// TIA Portal V15.1 export
// export: Created 2024-06-21T08:40:58.8620848Z, ExportSetting WithDefaults, DisplayName Totally Integrated Automation Portal, DisplayVersion V15.1 Update 5, DisplayName TIA Portal Openness, DisplayVersion V15.1 Update 5, DisplayName SINAMICS Startdrive Advanced, DisplayVersion V15.1, DisplayName G130, G150, S120, S150, SINAMICS MV, S210, DisplayVersion V15.1, DisplayName G110M, G120, G120C, G120D, G120P, DisplayVersion V15.1, DisplayName STEP 7 Professional, DisplayVersion V15.1 Update 5, DisplayName STEP 7 Safety, DisplayVersion V15.1, DisplayName WinCC Professional, DisplayVersion V15.1 Update 5, DisplayName SIMATIC Visualization Architect, DisplayVersion V15.1
FUNCTION_BLOCK "LPNIODiagNameS7-1500"   // FB2213, SCL
{ S7_Optimized_Access := 'TRUE' }
VERSION : 0.1
// stored: AutoNumber false, IsIECCheckEnabled false, IsRetainMemResEnabled false, MemoryReserve 100, SetENOAutomatically False, UDAEnableTagReadback false
   VAR_INPUT
      I_StartFillList { ExternalAccessible := 'False'; ExternalVisible := 'False'; ExternalWritable := 'False'} : Bool;
      I_LastDeviceNumber { ExternalAccessible := 'False'; ExternalVisible := 'False'; ExternalWritable := 'False'} : Int;   // Last Device of ProfiNet System
      I_HWIOSYSTEM { ExternalAccessible := 'False'; ExternalVisible := 'False'; ExternalWritable := 'False'} : HW_IOSYSTEM;   // HW ID ProfiNet System
   END_VAR
   VAR_OUTPUT
      O_Done { ExternalAccessible := 'False'; ExternalVisible := 'False'; ExternalWritable := 'False'} : Bool;
      O_Name { ExternalAccessible := 'False'; ExternalVisible := 'False'; ExternalWritable := 'False'} : Array[0..255] of String[25];
   END_VAR
   VAR_IN_OUT
      IO_DeviceExist : Array[0..255] of Bool;   // IO devices exist
      IO_GetStationName : Array[0..255] of String;   // Profinet Name
   END_VAR
   VAR
      Index { ExternalAccessible := 'False'; ExternalVisible := 'False'; ExternalWritable := 'False'} : Int;
      LastDeviceNumber { ExternalAccessible := 'False'; ExternalVisible := 'False'; ExternalWritable := 'False'} : Int;   // Last Device of ProfiNet System
      Done { ExternalAccessible := 'False'; ExternalVisible := 'False'; ExternalWritable := 'False'} : Bool;
      DoneDelay { ExternalAccessible := 'False'; ExternalVisible := 'False'; ExternalWritable := 'False'} : Bool;
      ReturnGetNameBusy { ExternalAccessible := 'False'; ExternalVisible := 'False'; ExternalWritable := 'False'} : Bool;   // Temp
      ReturnGetNameDone { ExternalAccessible := 'False'; ExternalVisible := 'False'; ExternalWritable := 'False'} : Bool;   // Temp
      ReturnGetNameError { ExternalAccessible := 'False'; ExternalVisible := 'False'; ExternalWritable := 'False'} : Bool;   // Temp
      ReturnGetNameLen { ExternalAccessible := 'False'; ExternalVisible := 'False'; ExternalWritable := 'False'} : DInt;   // Temp
      ReturnGetNameStatus { ExternalAccessible := 'False'; ExternalVisible := 'False'; ExternalWritable := 'False'} : Word;   // Temp
      GetNameInstance { ExternalAccessible := 'False'; ExternalVisible := 'False'; ExternalWritable := 'False'; S7_SetPoint := 'True'} : Get_Name;   // Get Name of Devices
      TimerDone { ExternalAccessible := 'False'; ExternalVisible := 'False'; ExternalWritable := 'False'; S7_SetPoint := 'True'} : TON_TIME;
      EdgeStartFillList { ExternalAccessible := 'False'; ExternalVisible := 'False'; ExternalWritable := 'False'; S7_SetPoint := 'True'} : R_TRIG;
   END_VAR
BEGIN
   #EdgeStartFillList(CLK := #I_StartFillList);

   IF #EdgeStartFillList.Q THEN
       #Done := False;
       #Index := 0;
   END_IF;

   #LastDeviceNumber := #I_LastDeviceNumber;
   IF #I_LastDeviceNumber < 1 THEN
       #LastDeviceNumber := 1;
   END_IF;
   IF #I_LastDeviceNumber > 254 THEN
       #LastDeviceNumber := 254;
   END_IF;


   #TimerDone(IN := #Done,
              PT := T#500ms,
              Q => #DoneDelay);

   IF (#I_StartFillList & NOT #Done) THEN
       #Index := #Index + 1;
       IF #IO_DeviceExist[#Index] THEN
           WHILE (#IO_DeviceExist[#Index] & NOT #ReturnGetNameDone) DO
               #GetNameInstance(LADDR := #I_HWIOSYSTEM,
                    STATION_NR := INT_TO_UINT(#Index),
                    DONE => #ReturnGetNameDone,
                    BUSY => #ReturnGetNameBusy,
                    ERROR => #ReturnGetNameError,
                    LEN => #ReturnGetNameLen,
                    STATUS => #ReturnGetNameStatus,
                    DATA := #IO_GetStationName[#Index]);
           END_WHILE;
           #ReturnGetNameDone := False;

           #O_Name[#Index] := #IO_GetStationName[#Index];
       END_IF;
       IF #Index = #LastDeviceNumber THEN
           #Done := True;
       END_IF;
   END_IF;

   #O_Done := #DoneDelay;
END_FUNCTION_BLOCK
